// TIA Portal V19 export
TYPE "Prg_Header"
// stored: Access Published
   STRUCT
      PrgNo : DInt;   // Program number
      PrgName : String[30];   // Program name
   END_STRUCT;
END_TYPE
